FUNCTION_BLOCK FB_FlowCommandFactory
VAR
END_VAR

METHOD CreateCompositeCommand : I_Command
VAR_INPUT
	invoker : I_CommandInvoker;
	description : STRING;
END_VAR
VAR	
	point : POINTER TO FB_CompositeCommand;
END_VAR
point := __NEW(FB_CompositeCommand(invoker := invoker, description := description));
CreateCompositeCommand := point^;
END_METHOD

METHOD CreateWaitCommand : I_Command
VAR_INPUT
	waitTime : TIME;
	description : STRING;
END_VAR
VAR	
	point : POINTER TO FB_WaitCommand;
END_VAR
point := __NEW(FB_WaitCommand(waitTime := waitTime, description := description));
CreateWaitCommand := point^;
END_METHOD

METHOD CreateWaitForConditionCommand : I_Command
VAR_INPUT
	condition : I_BoolValue;
	minWaitTime : TIME;
	maxWaitTime : TIME;
	description : STRING;
END_VAR
VAR	
	point : POINTER TO FB_WaitForConditionCommand;
END_VAR
point := __NEW(FB_WaitForConditionCommand(condition := condition, minWaitTime := minWaitTime, maxWaitTime := maxWaitTime, description := description));
CreateWaitForConditionCommand := point^;
END_METHOD

END_FUNCTION_BLOCK

(* stored: Version 1.1.0.1
   POU FB_FlowCommandFactory: Id {00868410-7edf-475a-b22e-9b46595a14e7}, SpecialFunc None
   Method CreateCompositeCommand: Id {a9d78103-dba1-460c-bdb1-e39f202e03fa}
   Method CreateWaitCommand: Id {95530303-1c50-4581-83d3-f1087474df25}
   Method CreateWaitForConditionCommand: Id {be81aff1-59f2-4e4e-a428-1d52f588ad1d} *)
